PROGRAM MAIN
VAR
	// Temp Sensor and Output variable created here.
	nTankTemp: REAL := 25;
	
	bHeaterON: BOOL := FALSE;
END_VAR

// Conditional IF statement detecting where Temperature is at
IF nTankTemp < 40.0 THEN
	bHeaterON := TRUE;
ELSIF nTankTemp > 60.0THEN
	bHeaterON := FALSE;
END_IF;

// Temperature changing in real time, being influenced by activation of heater
IF bHeaterON THEN
	nTankTemp := nTankTemp + 0.5;
ELSE
	nTankTemp := nTankTemp - 0.1;
END_IF;

END_PROGRAM

(* stored: Version 1.1.0.1, ProductVersion 3.1.4024.16
   POU MAIN: Id {e30d083e-3da6-47ae-8de8-8e47e27af3a0}, SpecialFunc None *)
